Staubli VAL3: getNum.pgx

program getNum(num& x_nNum (dimensions=1), num x_nEnd (dimensions=1))
begin
  sDataIn=""
  do
    nNbChar=sioGet(sioSocket,nData)
    if nNbChar>0 and nData!=x_nEnd
      sDataIn=sDataIn+chr(nData)
    endIf
  until nNbChar>0 and nData==x_nEnd
  sDataIn=toNum(sDataIn,x_nNum,bResult)
end
